PROGRAM P05_DeviceControl
VAR
	fbGreasing			:FB_Greaser;
	fbCamera			:FB_Handshake;
	fbRobot				:FB_Handshake;
	fbConveyor			:FB_Device;
	fbPickClamp			:FB_Device;
	fbPlaceClamp		:FB_Device;
	fbFeeder			:FB_Device;	
	fbIntakeBuffer		:FB_Stepper;
	fbOutletBuffer		:FB_Stepper;
END_VAR
VAR // added by the converter: edge detectors and wires of the graphical bodies
    _rt1, _rt2, _rt3, _rt4, _rt5 : R_TRIG;
    _ft1, _ft2, _ft3, _ft4 : F_TRIG;
END_VAR

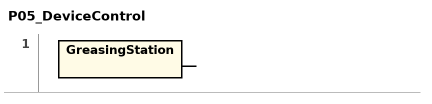
// NETWORK 1
GreasingStation();

ACTION Camera:
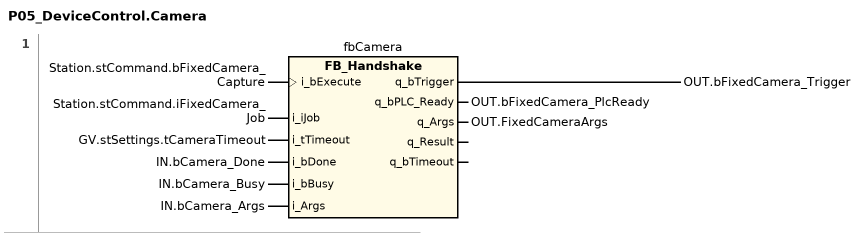
// NETWORK 1
_rt1(CLK := Station.stCommand.bFixedCamera_Capture);
fbCamera(
    i_bExecute := _rt1.Q,
    i_iJob := Station.stCommand.iFixedCamera_Job,
    i_tTimeout := GV.stSettings.tCameraTimeout,
    i_bDone := IN.bCamera_Done,
    i_bBusy := IN.bCamera_Busy,
    i_Args := IN.bCamera_Args,
    q_bPLC_Ready => OUT.bFixedCamera_PlcReady,
    q_Args => OUT.FixedCameraArgs); // FB_Handshake
OUT.bFixedCamera_Trigger := fbCamera.q_bTrigger;
END_ACTION

ACTION Conveyor:
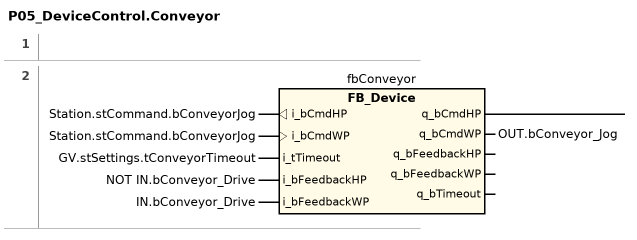
// NETWORK 1

// NETWORK 2
_ft1(CLK := Station.stCommand.bConveyorJog);
_rt2(CLK := Station.stCommand.bConveyorJog);
fbConveyor(
    i_bCmdHP := _ft1.Q,
    i_bCmdWP := _rt2.Q,
    i_tTimeout := GV.stSettings.tConveyorTimeout,
    i_bFeedbackHP := NOT IN.bConveyor_Drive,
    i_bFeedbackWP := IN.bConveyor_Drive,
    q_bCmdWP => OUT.bConveyor_Jog); // FB_Device
END_ACTION

ACTION Conveyor_PickClamp:
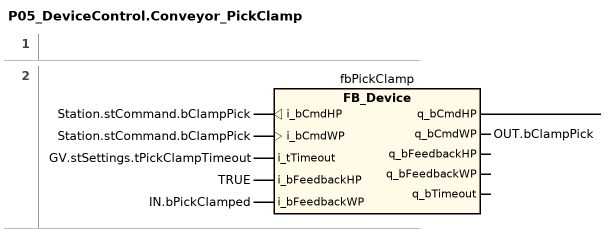
// NETWORK 1

// NETWORK 2
_ft2(CLK := Station.stCommand.bClampPick);
_rt3(CLK := Station.stCommand.bClampPick);
fbPickClamp(
    i_bCmdHP := _ft2.Q,
    i_bCmdWP := _rt3.Q,
    i_tTimeout := GV.stSettings.tPickClampTimeout,
    i_bFeedbackHP := TRUE,
    i_bFeedbackWP := IN.bPickClamped,
    q_bCmdWP => OUT.bClampPick); // FB_Device
END_ACTION

ACTION Conveyor_PlaceClamp:
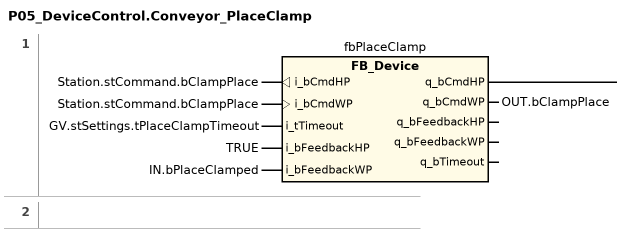
// NETWORK 1
_ft3(CLK := Station.stCommand.bClampPlace);
_rt4(CLK := Station.stCommand.bClampPlace);
fbPlaceClamp(
    i_bCmdHP := _ft3.Q,
    i_bCmdWP := _rt4.Q,
    i_tTimeout := GV.stSettings.tPlaceClampTimeout,
    i_bFeedbackHP := TRUE,
    i_bFeedbackWP := IN.bPlaceClamped,
    q_bCmdWP => OUT.bClampPlace); // FB_Device

// NETWORK 2
END_ACTION

ACTION Feeder:
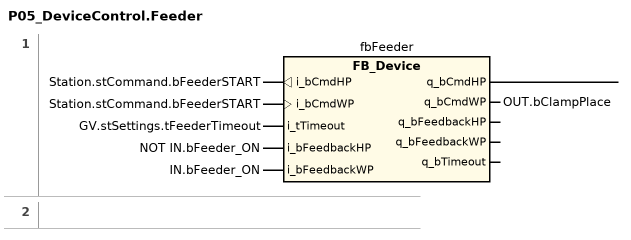
// NETWORK 1
_ft4(CLK := Station.stCommand.bFeederSTART);
_rt5(CLK := Station.stCommand.bFeederSTART);
fbFeeder(
    i_bCmdHP := _ft4.Q,
    i_bCmdWP := _rt5.Q,
    i_tTimeout := GV.stSettings.tFeederTimeout,
    i_bFeedbackHP := NOT IN.bFeeder_ON,
    i_bFeedbackWP := IN.bFeeder_ON,
    q_bCmdWP => OUT.bClampPlace); // FB_Device

// NETWORK 2
END_ACTION

ACTION GreasingStation:
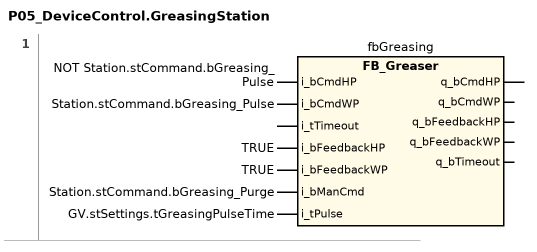
// NETWORK 1
fbGreasing(
    i_bCmdHP := NOT Station.stCommand.bGreasing_Pulse,
    i_bCmdWP := Station.stCommand.bGreasing_Pulse,
    i_bFeedbackHP := TRUE,
    i_bFeedbackWP := TRUE,
    i_bManCmd := Station.stCommand.bGreasing_Purge,
    i_tPulse := GV.stSettings.tGreasingPulseTime); // FB_Greaser
END_ACTION

ACTION IntakeBuffer:

END_ACTION

ACTION OuletBuffer:
// NETWORK 1
END_ACTION

ACTION Robot:
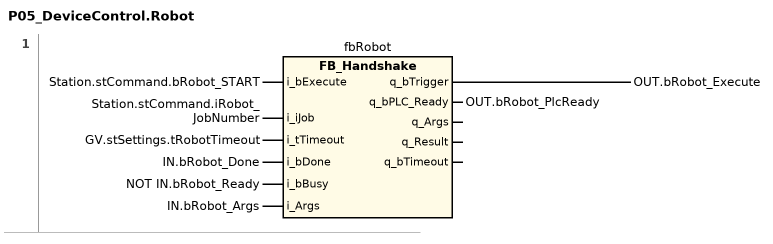
// NETWORK 1
fbRobot(
    i_bExecute := Station.stCommand.bRobot_START,
    i_iJob := Station.stCommand.iRobot_JobNumber,
    i_tTimeout := GV.stSettings.tRobotTimeout,
    i_bDone := IN.bRobot_Done,
    i_bBusy := NOT IN.bRobot_Ready,
    i_Args := IN.bRobot_Args,
    q_bPLC_Ready => OUT.bRobot_PlcReady); // FB_Handshake
OUT.bRobot_Execute := fbRobot.q_bTrigger;
END_ACTION

END_PROGRAM

(* stored: Version 1.1.0.1
   POU P05_DeviceControl: Id {0de36414-366b-4231-b48a-58e7f43e3efd}, SpecialFunc None
   Action Camera: Id {7d919d6a-e71b-49c3-a19c-19022d089980}
   Action Conveyor: Id {29d9be05-e312-44fb-85cc-3aa1c048611c}
   Action Conveyor_PickClamp: Id {9c307688-40ba-4500-84b7-c9fa1af78e3b}
   Action Conveyor_PlaceClamp: Id {64641713-c2ea-42f5-892a-9e14c3cffec9}
   Action Feeder: Id {01a5c520-470b-444b-aa82-bb5d64c9ac87}
   Action GreasingStation: Id {a8fdd751-43fe-4fd9-a0c2-7cb896dc2e03}
   Action IntakeBuffer: Id {ed317e41-37e2-49fc-9d3f-cb6098ef64af}
   Action OuletBuffer: Id {6cda1e91-81b8-4d6b-abc0-4d2296ad1410}
   Action Robot: Id {105d1f1c-6cd5-47c9-8253-4feb34d6911a} *)
